INTERFACE ITF_Robot EXTENDS ITF_BaseComponent

METHOD disable : BOOL
VAR_INPUT
END_VAR
END_METHOD

METHOD disableVelocityOverride : BOOL
VAR_INPUT
END_VAR
END_METHOD

METHOD enable : BOOL
VAR_INPUT
END_VAR
END_METHOD

METHOD enableVelocityOverride : BOOL
VAR_INPUT
END_VAR
END_METHOD

METHOD estop : BOOL
VAR_INPUT
END_VAR
END_METHOD

METHOD M_AUTO : BOOL
VAR_INPUT
END_VAR
END_METHOD

METHOD M_MAN : BOOL
VAR_INPUT
END_VAR
END_METHOD

METHOD MC_ChangeSpeedOverride : INT
VAR_INPUT
	factor: REAL;
END_VAR
END_METHOD

METHOD MC_MoveAxesAbsolute : BOOL
VAR_INPUT
	target: stTarget3D;
END_VAR
END_METHOD

METHOD MC_MoveAxesRelative : BOOL
VAR_INPUT
	axes: ARRAY[1..6] OF FB_Axis;
	offsets: ARRAY[1..6] OF REAL;
END_VAR
END_METHOD

METHOD MC_MoveLinearAbsolute : BOOL
VAR_INPUT
	target: stTarget3D;
END_VAR
END_METHOD

METHOD PUBLIC MC_ReadActualVelocity : stPose
VAR_INPUT
END_VAR
VAR

END_VAR
END_METHOD

METHOD PUBLIC MC_ReadAnalogInput : LREAL
VAR_INPUT
	input : INT;
END_VAR
END_METHOD

METHOD PUBLIC MC_ReadDigitalInput : BOOL
VAR_INPUT
	input : INT;
END_VAR
END_METHOD

METHOD PUBLIC MC_SetDigitalOutput : BOOL
VAR_INPUT
	output : INT;
	value : BOOL;
END_VAR
END_METHOD

METHOD PUBLIC MC_SetOperationMode : BOOL
VAR_INPUT
	mode: eMode;
END_VAR
END_METHOD

METHOD stop : BOOL
VAR_INPUT
END_VAR
END_METHOD

END_INTERFACE

(* stored: Version 1.1.0.1, ProductVersion 3.1.4026.18
   Itf ITF_Robot: Id {a6d29cf6-e144-4e1d-bf83-e7b2be10a693}
   Method disable: Id {1f5c5c05-2dcb-40b6-85b7-e14de76733ca}
   Method disableVelocityOverride: Id {1643e2ed-a195-4fb9-bcc2-d0e7b52e61fb}
   Method enable: Id {0f3f76ce-0c24-431f-b0cb-d24dc0415a91}
   Method enableVelocityOverride: Id {a219643f-8e25-47f8-b4f4-e2335d3e6ead}
   Method estop: Id {6bd7f640-7106-49dd-a5cd-96054e8ed6ff}
   Method M_AUTO: Id {4a5f6fe2-c0ac-4a0a-ac11-a7823ebd0b5f}
   Method M_MAN: Id {bd189bc6-367b-4937-84f7-9d3aaa9bc52d}
   Method MC_ChangeSpeedOverride: Id {ab6ffcb5-7287-4c7e-a668-cb65a48c6fd6}
   Method MC_MoveAxesAbsolute: Id {3f8dd969-4475-4859-99c9-640266c99491}
   Method MC_MoveAxesRelative: Id {622605cf-64f8-437c-8219-d922cc2e68c1}
   Method MC_MoveLinearAbsolute: Id {e8bb4eaf-5055-49b0-a341-8aba2f3636ff}
   Method MC_ReadActualVelocity: Id {4f6a0ffe-d696-474a-b5be-142c98ad027d}
   Method MC_ReadAnalogInput: Id {13341557-e12d-40d5-bfb4-957c78230509}
   Method MC_ReadDigitalInput: Id {4c842e7c-5020-4038-a32e-d6559a620f63}
   Method MC_SetDigitalOutput: Id {06120d26-3887-4b04-8b2c-a46eb00a3b04}
   Method MC_SetOperationMode: Id {bec57ab4-062c-4029-a3ba-e9e22a17f741}
   Method stop: Id {3ff1b608-cbee-4153-8537-8c5ca10ccc31} *)
